(*
Abstract function block providing an :attr:`Input` property for single-input
controller toolbox components.

Concrete implementations read from ``_fInput`` to consume the signal written
by the caller.

.. note::
   Direct calls to this function block are not permitted (``no_explicit_call``).
   Extend it and call the derived block instead.
*)
{attribute 'no_explicit_call' := 'direct call for this function block is not allowed'}
FUNCTION_BLOCK ABSTRACT FB_SiComponent
IMPLEMENTS I_SiComponent
VAR
    _fInput : LREAL;
END_VAR

(* Gets or sets the input to the component.*)
PROPERTY Input : LREAL
GET
Input := THIS^._fInput;
END_GET
SET
THIS^._fInput := Input;
END_SET
END_PROPERTY

END_FUNCTION_BLOCK

(* stored: Version 1.1.0.1, ProductVersion 3.1.4024.15
   POU FB_SiComponent: Id {af4e3e06-6e07-4751-bb2e-628529d86b2a}, SpecialFunc None
   Property Input: Id {3fa3a351-fd3a-4829-a136-b7ae0143ce13}
   Get Get: Id {30895f99-b4e4-4b92-8f97-adbaf61238bc}
   Set Set: Id {fa1deed6-2ff9-47a7-a459-3445f9fce041} *)
